SYSTEM Example
  (* Version 1.0, 2007-08-28, Goran Cengic, Chalmers *)
  DEVICE Test Device : DeviceType_not_used
    RESOURCE TestResource : ResourceType_not_used
      FBS
        restart : E_RESTART;
        stop : E_STOP;
        split : E_SPLIT2;
        rend : E_REND;
        prod1 : Product;
        prod2 : Product;
        res1 : Resource;
        res2 : Resource;
        res3 : Resource;
      END_FBS
      EVENT_CONNECTIONS
        restart.COLD TO split.EI;
        split.EO1 TO prod1.make;
        split.EO2 TO prod2.make;
        prod1.takeR1 TO res1.take1;
        prod1.takeR2 TO res2.take1;
        prod1.takeR3 TO res3.take1;
        prod1.processR1 TO res1.process1;
        prod1.processR2 TO res2.process1;
        prod1.processR3 TO res3.process1;
        prod1.releaseR1 TO res1.release1;
        prod1.releaseR2 TO res2.release1;
        prod1.releaseR3 TO res3.release1;
        res1.taken1 TO prod1.gotR1;
        res2.taken1 TO prod1.gotR2;
        res3.taken1 TO prod1.gotR3;
        res1.processed1 TO prod1.processedR1;
        res2.processed1 TO prod1.processedR2;
        res3.processed1 TO prod1.processedR3;
        prod2.takeR1 TO res1.take2;
        prod2.takeR2 TO res2.take2;
        prod2.takeR3 TO res3.take2;
        prod2.processR1 TO res1.process2;
        prod2.processR2 TO res2.process2;
        prod2.processR3 TO res3.process2;
        prod2.releaseR1 TO res1.release2;
        prod2.releaseR2 TO res2.release2;
        prod2.releaseR3 TO res3.release2;
        res1.taken2 TO prod2.gotR1;
        res2.taken2 TO prod2.gotR2;
        res3.taken2 TO prod2.gotR3;
        res1.processed2 TO prod2.processedR1;
        res2.processed2 TO prod2.processedR2;
        res3.processed2 TO prod2.processedR3;
        prod1.done TO rend.EI1;
        prod2.done TO rend.EI2;
        rend.EO TO stop.STOP;
      END_CONNECTIONS
      DATA_CONNECTIONS
        1 TO prod1.product;
        2 TO prod2.product;
        1 TO res1.capacity;
        1 TO res2.capacity;
        1 TO res3.capacity;
      END_CONNECTIONS
    END_RESOURCE
  END_DEVICE
END_SYSTEM
(* other elements stored in the file *)
(* Product 1 *)
(* Product 2 *)
